TYPE EN_SequenceMode :
(
	SequenceModeNormal := 0,
	SequenceModeStep,
	SequenceModeBreak
);
END_TYPE

(* stored: Version 1.1.0.1, ProductVersion 3.1.0.36
   DUT EN_SequenceMode: Id {eceb5ad1-87f6-464a-bdaf-0cd532b18bd0} *)
